// TIA Portal V21 export
DATA_BLOCK "AiDb"   // DB108
// stored: AutoNumber false, InstanceOfName AiFb, InstanceOfType FB
"AiFb"
   // VAR
   //    Ai01 { S7_SetPoint := 'True'} : "FB:Analog_Scaling";   // NfcoLineTemp(Ticr01)
   //    Ai02 { S7_SetPoint := 'True'} : "FB:Analog_Scaling";   // VfcoLineTemp(Ticr02)
   //    Ai03 { S7_SetPoint := 'True'} : "FB:Analog_Scaling";   // AiSpare01
   //    Ai04 { S7_SetPoint := 'True'} : "FB:Analog_Scaling";   // AiSpare02
   //    Ai05 { S7_SetPoint := 'True'} : "FB:Analog_Scaling";   // AiSpare03
   //    Ai06 { S7_SetPoint := 'True'} : "FB:Analog_Scaling";   // Pf01InLineTemp(Ticr06)
   //    Ai07 { S7_SetPoint := 'True'} : "FB:Analog_Scaling";   // Pf02InLineTemp(Ticr07)
   //    Ai08 { S7_SetPoint := 'True'} : "FB:Analog_Scaling";   // Pf02OutLineTemp(Ticr08)
   //    Ai09 { S7_SetPoint := 'True'} : "FB:Analog_Scaling";   // PtlDrainTemp(Ticr09)
   //    Ai10 { S7_SetPoint := 'True'} : "FB:Analog_Scaling";   // VesselTemp(Ticr10)
   //    Ai11 { S7_SetPoint := 'True'} : "FB:Analog_Scaling";   // VesselPressure(Picr01)
   //    Ai12 { S7_SetPoint := 'True'} : "FB:Analog_Scaling";   // VesselRclLine(Picr02)
   //    Ai13 { S7_SetPoint := 'True'} : "FB:Analog_Scaling";   // Pf01OutLinePressure(Picr03)
   //    Ai14 { S7_SetPoint := 'True'} : "FB:Analog_Scaling";   // Pf02OutLinePressure(Picr04)
   //    Ai15 { S7_SetPoint := 'True'} : "FB:Analog_Scaling";   // ProcessDrainConductivity
   //    Ai16 { S7_SetPoint := 'True'} : "FB:Analog_Scaling";   // AiSpare04
   //    Ai17 { S7_SetPoint := 'True'} : "FB:Analog_Scaling";   // AiSpare05
   //    Ai18 { S7_SetPoint := 'True'} : "FB:Analog_Scaling";   // AiSpare06
   //    Ai19 { S7_SetPoint := 'True'} : "FB:Analog_Scaling";   // AiSpare07
   //    Ai20 { S7_SetPoint := 'True'} : "FB:Analog_Scaling";   // AiSpare08
   //    Ai21 { S7_SetPoint := 'True'} : "FB:Analog_Scaling";   // AiSpare09
   //    Ai22 { S7_SetPoint := 'True'} : "FB:Analog_Scaling";   // AiSpare10
   //    Ai23 { S7_SetPoint := 'True'} : "FB:Analog_Scaling";   // AiSpare11
   //    Ai24 { S7_SetPoint := 'True'} : "FB:Analog_Scaling";   // AiSpare12
   // END_VAR
BEGIN
   Ai01.AlmHighLimit := 150.0;
   Ai01.AlmLowlimit := -15.0;
   Ai01.HighRange := 150.0;
   Ai01.LowRange := -15.0;
   Ai02.AlmHighLimit := 150.0;
   Ai02.AlmLowlimit := -15.0;
   Ai02.HighRange := 150.0;
   Ai02.LowRange := -15.0;
   Ai02.LowAlarmStatus := 0;
   Ai03.AlmHighLimit := 150.0;
   Ai03.AlmLowlimit := -15.0;
   Ai03.HighRange := 150.0;
   Ai03.LowRange := -15.0;
   Ai04.AlmHighLimit := 150.0;
   Ai04.AlmLowlimit := -15.0;
   Ai04.HighRange := 150.0;
   Ai04.LowRange := -15.0;
   Ai04.LowAlarmStatus := 0;
   Ai05.AlmHighLimit := 150.0;
   Ai05.AlmLowlimit := -15.0;
   Ai05.HighRange := 150.0;
   Ai05.LowRange := -15.0;
   Ai05.LowAlarmStatus := 0;
   Ai06.AlmHighLimit := 150.0;
   Ai06.AlmLowlimit := -15.0;
   Ai06.HighRange := 150.0;
   Ai06.LowRange := -15.0;
   Ai06.LowAlarmStatus := 0;
   Ai07.AlmHighLimit := 150.0;
   Ai07.AlmLowlimit := -15.0;
   Ai07.HighRange := 150.0;
   Ai07.LowRange := -15.0;
   Ai08.AlmHighLimit := 150.0;
   Ai08.AlmLowlimit := -15.0;
   Ai08.HighRange := 150.0;
   Ai08.LowRange := -15.0;
   Ai09.AlmHighLimit := 150.0;
   Ai09.AlmLowlimit := -15.0;
   Ai09.HighRange := 150.0;
   Ai09.LowRange := -15.0;
   Ai10.AlmHighLimit := 150.0;
   Ai10.AlmLowlimit := -15.0;
   Ai10.HighRange := 150.0;
   Ai10.LowRange := -15.0;
   Ai11.AlmHighLimit := 5.0;
   Ai11.AlmLowlimit := -1.0;
   Ai11.HighRange := 5.0;
   Ai11.LowRange := -1.0;
   Ai12.AlmHighLimit := 5.0;
   Ai12.AlmLowlimit := -1.0;
   Ai12.HighRange := 5.0;
   Ai12.LowRange := -1.0;
   Ai13.AlmHighLimit := 5.0;
   Ai13.AlmLowlimit := -1.0;
   Ai13.HighRange := 5.0;
   Ai13.LowRange := -1.0;
   Ai14.HighRange := 5.0;
   Ai14.LowRange := -1.0;
   Ai15.HighRange := 100.0;
   Ai15.LowRange := 0.0;
END_DATA_BLOCK
